{attribute 'linkalways'} 
{attribute 'no_explicit_call' := 'This FB is a CLASS and must be accessed using methods or properties'}
{attribute 'enable_dynamic_creation'}
FUNCTION_BLOCK FINAL AND_BYTE EXTENDS Node
VAR
	in1 : _BYTE(0);
	in2 : _BYTE(0);
	out : _BYTE(0);
END_VAR

METHOD PUBLIC Clone : I_Node
VAR
	pNode : POINTER TO AND_BYTE;
END_VAR
pNode := __NEW(AND_BYTE);
Clone := pNode^;
END_METHOD

METHOD FB_init : BOOL
VAR_INPUT
	bInitRetains : BOOL; // if TRUE, the retain variables are initialized (warm start / cold start)
	bInCopyCode : BOOL;  // if TRUE, the instance afterwards gets moved into the copy code (online change)
END_VAR
AddInput('in1',THIS^.in1);
AddInput('in2',THIS^.in2);
AddOutput('out', THIS^.out);
END_METHOD

METHOD PROTECTED OnExecute
VAR
END_VAR
out.Value := in1.Value AND in2.Value;
END_METHOD

END_FUNCTION_BLOCK

(* stored: Version 1.1.0.1, ProductVersion 3.1.4024.15
   POU AND_BYTE: Id {bfd6e258-c49c-4591-94cf-f67c7be61f74}, SpecialFunc None
   Folder Constructor: Id {452d622f-67e0-4dd0-9af0-53e1d05cf4e7}
   Method Clone: Id {5d8f31c7-655c-49e9-a554-d5dd7050f2e1}
   Method FB_init: Id {361eef50-7a89-4bc6-9b5d-20e7a5398b63}
   Method OnExecute: Id {ee74ba58-58b4-47ba-8950-7f19c5757b47} *)
